FUNCTION_BLOCK FB_PneuCyl_3Pos EXTENDS FB_Base
VAR_INPUT
END_VAR
VAR_OUTPUT
END_VAR
VAR
	
	fbBottomOut												: FB_Output					  (GVL_Customer.C_Name_PneuCylBottomOut,
																													 GVL_Customer.C_ID_PneuCylBottomOut
																											  	);
																														
	fbTopOut													: FB_Output					  (GVL_Customer.C_Name_PneuCylTopOut,
																													 GVL_Customer.C_ID_PneuCylTopOut
																											  	);
	
	fbBouttomIn												: FB_Input					  (GVL_Customer.C_Name_PneuCylMiddleIn,
																													 GVL_Customer.C_ID_PneuCylMiddleIn
																											  	);

	fbTopIn 													: FB_Input					  (GVL_Customer.C_Name_PneuCylMiddleIn,
																													 GVL_Customer.C_ID_PneuCylMiddleIn
																											  	);
																												
	fbMiddleIn												: FB_Input					  (GVL_Customer.C_Name_PneuCylMiddleIn,
																													 GVL_Customer.C_ID_PneuCylMiddleIn
																											  	);
																													
																													
END_VAR

//================== Must!!
SUPER^();  
IF NOT Enable THEN RETURN; END_IF;

//FB_Init ist immer implizit verfügbar und wird primär für die Initialisierung verwendet.
//Der Rückgabewert wird nicht ausgewertet. Für gezielte Einflussnahme können Sie
//die Methoden explizit deklarieren und darin mit dem Standard-Initialisierungscode 
//zusätzlichen Code bereitstellen. Sie können den Rückgabewert auswerten.
METHOD FB_Init: BOOL
VAR_INPUT    
	bInitRetains					: BOOL; 					// TRUE: Die Retain-Variablen werden initialisiert (Reset warm / Reset kalt)    
	bInCopyCode						: BOOL;  					// TRUE: Die Instanz wird danach in den Kopiercode kopiert (Online-Change)
	
	I_Name                : STRING;         //  Name
	I_ID                  : UINT;            // ID
END_VAR
END_METHOD

METHOD mCallBottom : E_CmdState
VAR_INPUT
	I_bExecute			 : BOOL;
END_VAR
// No command requested.
IF NOT I_bExecute 
	THEN
    mCallBottom  := E_CmdState.Idle;
    RETURN;
END_IF

// Command cylinder to top.
// To Bottom=True, To Top=False.

fbBottomOut.bBoolValue 	:= TRUE;
fbTopOut.bBoolValue   	:= FALSE;

// Wait until top sensor is active.
IF fbBouttomIn.bBoolValue 
	THEN
		mCallBottom 	:= E_CmdState.Succeeded;
ELSE
    mCallBottom 	:= E_CmdState.Busy;
END_IF
END_METHOD

METHOD mCallMiddle : E_CmdState
VAR_INPUT
	I_bExecute			 : BOOL;
END_VAR
// No command requested.
IF NOT I_bExecute 
	THEN
    mCallMiddle    := E_CmdState.Idle;
    RETURN;
END_IF

// Command cylinder to Middle.
// To Bottom=False, To Top=False.
fbBottomOut.bBoolValue 	   := FALSE;
fbTopOut.bBoolValue    		 := FALSE;

// Wait until top sensor is active.
IF fbMiddleIn.bIAT_bHardwareLink 
	THEN
		mCallMiddle 	 := E_CmdState.Succeeded;
ELSE
    mCallMiddle 	 := E_CmdState.Busy;
END_IF
END_METHOD

METHOD mCallTop : E_cmdState
VAR_INPUT
	I_bExecute		: BOOL;
END_VAR
// No command requested.
IF NOT I_bExecute 
	THEN
    mCallTop       := E_CmdState.Idle;
    RETURN;
END_IF

// Command cylinder to top.
// ToBottom=FALSE, ToTop=TRUE.
fbBottomOut.bBoolValue 		 := FALSE;
fbTopOut.bBoolValue    	   := TRUE;

// Wait until top sensor is active.
IF fbTopIn.bBoolValue 
	THEN
		mCallTop 			 := E_CmdState.Succeeded;
ELSE
    mCallTop 			 := E_CmdState.Busy;
END_IF
END_METHOD

END_FUNCTION_BLOCK

(* stored: Version 1.1.0.1, ProductVersion 3.1.4026.18
   POU FB_PneuCyl_3Pos: Id {539861d2-79e9-47d0-b2b0-f4891b2941c6}, SpecialFunc None
   Folder 01 Properties: Id {7f9f3ab8-59ae-4eca-a2d4-19e93fc901fc}
   Folder 02 Methodes: Id {fcbe53fd-f5c0-4865-babd-f6fd9d39dfd6}
   Folder 100 CmdExecute: Id {2638535f-0cf6-460e-9dfd-d9fc56172997}
   Method FB_Init: Id {8d364b46-6db2-4a0b-a3fd-36a170ec67fd}
   Method mCallBottom: Id {20d57b03-bf1d-4ff1-b123-9c04c00c3255}
   Method mCallMiddle: Id {4fbc886a-155d-41b4-b539-a6a894d01499}
   Method mCallTop: Id {024c0db2-8530-4e9f-8ed6-a6d408c8fbd6} *)
